SUBAPPLICATION mapping (* Subapplication Type *)
  (* Standard: 61499-2 *)
  (* Version 1.0, 2023-02-19, franz *)
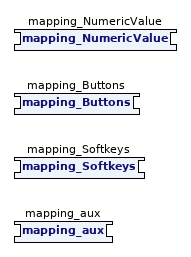
  SUBAPPS
    mapping_NumericValue : mapping_NumericValue;
    mapping_Softkeys : mapping_Softkeys;
    mapping_Buttons : mapping_Buttons;
    mapping_aux : mapping_aux;
  END_SUBAPPS
END_SUBAPPLICATION
